FUNCTION_BLOCK Logger IMPLEMENTS ILogger
VAR_INPUT
END_VAR
VAR_OUTPUT
	ipResultMessage : I_TcMessage := fbResult;
END_VAR
VAR
	fbResult : FB_TcMessage;
	fbSource : FB_TcSourceInfo;
	
	hrLastInternalError : HRESULT;	
END_VAR

METHOD Debug
VAR_INPUT
	message	: STRING;
END_VAR
VAR
	hr : HRESULT;
END_VAR
hr := fbResult.CreateEx(TC_EVENTS.EventLoggerPlc.PlcEventDebug, ipSourceInfo:=fbSource);
Write(message, hr);
END_METHOD

METHOD Error
VAR_INPUT
	message	: STRING;
END_VAR
VAR
	hr : HRESULT;
END_VAR
hr := fbResult.CreateEx(TC_EVENTS.EventLoggerPlc.PlcEventError, ipSourceInfo:=fbSource);
Write(message, hr);
END_METHOD

METHOD Fatal
VAR_INPUT
	message	: STRING;
END_VAR
VAR
	hr : HRESULT;
END_VAR
hr := fbResult.CreateEx(TC_EVENTS.EventLoggerPlc.PlcEventFatal, ipSourceInfo:=fbSource);
Write(message, hr);
END_METHOD

METHOD Information
VAR_INPUT
	message	: STRING;
END_VAR
VAR
	hr : HRESULT;
END_VAR
hr := fbResult.CreateEx(TC_EVENTS.EventLoggerPlc.PlcEventInformation, ipSourceInfo:=fbSource);
Write(message, hr);
END_METHOD

METHOD Verbose
VAR_INPUT
	message	: STRING;
END_VAR
VAR
	hr : HRESULT;
END_VAR
hr := fbResult.CreateEx(TC_EVENTS.EventLoggerPlc.PlcEventVerbose, ipSourceInfo:=fbSource);
Write(message, hr);
END_METHOD

METHOD Warning
VAR_INPUT
	message	: STRING;
END_VAR
VAR
	hr : HRESULT;
END_VAR
hr := fbResult.CreateEx(TC_EVENTS.EventLoggerPlc.PlcEventWarning, ipSourceInfo:=fbSource);
Write(message, hr);
END_METHOD

METHOD PRIVATE Write
VAR_INPUT
	message : STRING;
	handle : HRESULT;
END_VAR
fbResult.ipArguments.Clear().AddString(message);

IF fbResult.eSeverity >= TcEventSeverity.Verbose THEN
	handle := fbResult.Send(0);
	IF FAILED(handle) THEN
		hrLastInternalError := handle;
	END_IF
END_IF
END_METHOD

END_FUNCTION_BLOCK

(* stored: Version 1.1.0.1, ProductVersion 3.1.4024.3
   POU Logger: Id {be1f4ad8-0ce5-4bde-aeca-b5f947db7668}, SpecialFunc None
   Method Debug: Id {c400de67-60eb-43d6-b271-b20e176ef72c}
   Method Error: Id {bcf18f5c-f01e-4da0-930b-a08e3759103d}
   Method Fatal: Id {cfd1644f-ce03-4ef9-a353-fe517e29affa}
   Method Information: Id {4cc4e622-0cb9-4ccb-8de0-dd2c5c6c72f1}
   Method Verbose: Id {1b73ddbb-5494-4163-817c-b03176bca5b8}
   Method Warning: Id {bdaee934-5679-4dc1-98bd-525abbaa460d}
   Method Write: Id {8d4fd826-cd66-4f89-817a-a0df49536ee7} *)
